FUNCTION_BLOCK WatchdogCheckExtension EXTENDS Extension
VAR
	watchdogAlarm : FunctionFailedAlarm(THIS^);
	watchdogTimeInUs : _DINT(10000000); // default 10s
	hResult : HRESULT;
END_VAR

METHOD FB_init : BOOL
VAR_INPUT
	bInitRetains : BOOL; // if TRUE, the retain variables are initialized (warm start / cold start)
	bInCopyCode : BOOL;  // if TRUE, the instance afterwards gets moved into the copy code (online change)
	Name : T_MAXSTRING;
	Parent : I_HostExtensions;
END_VAR
AddParameter('watchdogTimeInUs', watchdogTimeInUs);
END_METHOD

METHOD PUBLIC Start
VAR_INPUT
END_VAR
watchdogAlarm.Clear();

IF watchdogTimeInUs.Value = 0 THEN
	RETURN;
END_IF

hResult := F_VN_StartRelWatchdog(watchdogTimeInUs.Value, S_OK);
END_METHOD

METHOD PUBLIC Stop
VAR_INPUT
END_VAR
hresult := F_VN_StopWatchdog(
	hrStartWatchdog := hresult);

IF FAILED(hresult) THEN
	watchdogAlarm.Raise('Watchdog', hresult);
END_IF
END_METHOD

END_FUNCTION_BLOCK

(* stored: Version 1.1.0.1, ProductVersion 3.1.4026.18
   POU WatchdogCheckExtension: Id {c414888c-294b-00e8-26d1-35c6bbb6ba50}, SpecialFunc None
   Folder Constructor: Id {0f50eb21-d707-0d4c-2985-38486fd76614}
   Method FB_init: Id {7d855a95-77ef-076b-3bc3-51b2e694fba3}
   Method Start: Id {3c805fc1-4eb4-0160-060f-6a55c0259a43}
   Method Stop: Id {1d99623e-567c-0206-29ce-9507611054ae} *)
